FUNCTION_BLOCK Conveyor EXTENDS BaseComponent
VAR_INPUT
END_VAR
VAR_OUTPUT
END_VAR
VAR
	Motor : Motor;
END_VAR

METHOD METH_ConveyorBackward : BOOL
VAR_INPUT
END_VAR
Motor.ACT_TurnCounterclockwise();
END_METHOD

METHOD METH_ConveyorForward : BOOL
VAR_INPUT
END_VAR
Motor.ACT_TurnClockwise();
END_METHOD

METHOD METH_ConveyorStop : BOOL
VAR_INPUT
END_VAR
Motor.ACT_Stop();
END_METHOD

END_FUNCTION_BLOCK

(* stored: Version 1.1.0.1, ProductVersion 3.1.4024.4
   POU Conveyor: Id {8bf5544b-891e-499c-b4aa-85e5ed9acb50}, SpecialFunc None
   Method METH_ConveyorBackward: Id {50d9e013-3266-480b-83c7-2956ddadd8f9}
   Method METH_ConveyorForward: Id {b845516b-21a4-4031-a47c-f1c30b945be8}
   Method METH_ConveyorStop: Id {b3690ca6-57fb-4e40-917a-ad9f2b4a72ca} *)
